TYPE ST_EL1004 :
STRUCT
	Inputs	AT %I*	: ARRAY[0..3] OF BOOL;
END_STRUCT
END_TYPE

(* stored: Version 1.1.0.1, ProductVersion 3.1.4024.6
   DUT ST_EL1004: Id {384e0d28-ef56-4123-81da-c6a1eea42fcd} *)
